Staubli VAL3: _resizeData.pgx

program _resizeData(num x_nSizeTxt, num x_nSizeLbl)
begin
  // Resize numerics
  resize(nLblPosX,1,x_nSizeLbl)
  resize(nLblPosY,1,x_nSizeLbl)
  resize(nTxtMaxVal,1,x_nSizeTxt)
  resize(nTxtMinVal,1,x_nSizeTxt)
  resize(nTxtPosX,1,x_nSizeTxt)
  resize(nTxtPosY,1,x_nSizeTxt)
end
